PROGRAM MAIN
VAR
END_VAR

//One

//Two

END_PROGRAM

(* stored: Version 1.1.0.1, ProductVersion 3.1.4024.9
   POU MAIN: Id {9c522426-348a-4e47-ad37-3efe9051d437}, SpecialFunc None *)
